// TIA Portal V16 export
// export: Created 2024-04-19T15:29:40.4784353Z, ExportSetting WithDefaults, DisplayName Totally Integrated Automation Portal, DisplayVersion V16 Update 6, DisplayName TIA Portal Version Control Interface, DisplayVersion V16 Update 2, DisplayName TIA Portal Openness, DisplayVersion V16 Update 6, DisplayName TIA Portal Test Suite Advanced, DisplayVersion V16, DisplayName SINAMICS Startdrive Advanced, DisplayVersion V16 Update 5, DisplayName SINAMICS Startdrive G130, G150, S120, S150, SINAMICS MV, S210, DisplayVersion V16 Update 5, DisplayName SINAMICS Startdrive G110M, G120, G120C, G120D, G120P, G115D, DisplayVersion V16 Update 5, DisplayName STEP 7 Professional, DisplayVersion V16 Update 6, DisplayName STEP 7 Safety, DisplayVersion V16, DisplayName WinCC Advanced, DisplayVersion V16 Update 6
TYPE "SCA_beltConveyor"
// stored: IsFailsafeCompliant false
   STRUCT
      IO { S7_SetPoint := 'True'} : "SCA_slatConveyor_IO";
      Status { S7_SetPoint := 'True'} : "SCA_Status";
      Control { S7_SetPoint := 'True'} : "RMP_UDT_CONTROL";
      Frq { S7_SetPoint := 'True'} : "RMP_BIF_FRQ_SPD";
      Drive { S7_SetPoint := 'True'} : "RMP_BIF_FRQ_SPD";
      Interlock { S7_SetPoint := 'True'} : "SCA_Interlock";
      Flags { S7_SetPoint := 'True'} : "SCA_Flags";
      Device_name { S7_SetPoint := 'True'} : String[40];
   END_STRUCT;
END_TYPE
